% RSLogix 500 project alarm_count_live.RSS, saved by version 8.30.00.16 %
PROJECT "UNTITLED"    % processor: Bul.1763 MicroLogix 1100 Series B %

PROGRAM FILES
  LAD 2 "MAIN"  4 rungs
  LAD 3 "SUB_AND"  6 rungs
  LAD 4 "PARALLEL"  12 rungs
  LAD 5 "XIC_BRUTEF"  3 rungs
  LAD 6 "LOOKUPBYTE"  5 rungs
  LAD 7 "WRITE_BITS"  5 rungs
  LAD 255 "BITSPRBYTE"  5 rungs

DATA FILES
  O0 OUTPUT  4 elements
  I1 INPUT  6 elements
  S2 STATUS  66 elements
  B3 BINARY  3 elements
  T4 TIMER  11 elements
  C5 COUNTER  1 elements
  R6 CONTROL  1 elements
  N7 INTEGER  10 elements
  F8 FLOAT  4 elements
  L9 LONG_DATA  12 elements
  N10 BITSPRBYTE  256 elements
  L11 LONG_MASKS  12 elements
  L100 CONTRLTIME  256 elements
  L101 SUBANDTIME  256 elements
  L102 PARLLLTIME  256 elements
  L103 XIC_TIME  256 elements
  L104 LOOKUPTIME  256 elements

LADDER 2 "MAIN"
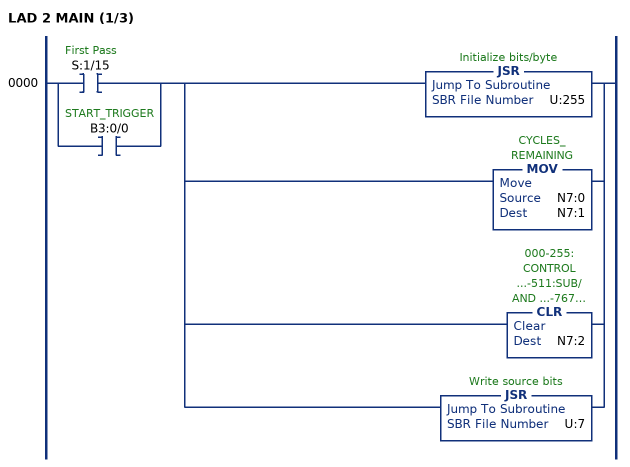
% Rung: 0 %
SOR BST XIC S:1/15 NXB XIC B3:0/0 BND BST JSR U:255 NXB MOV N7:0 N7:1 NXB CLR N7:2 NXB JSR U:7 BND EOR
%   S:1/15  "First Pass" %
%   B3:0/0  START_TRIGGER %
%   U:255  "Initialize bits/byte" %
%   N7:0  TEST_CYCLES %
%   N7:1  CYCLES_REMAINING %
%   N7:2  WHICH  "000-255:CONTROL ...-511:SUB/AND ...-767:PARALLEL ...-1023:XIC ...-1279:LOOKUP_BYTE" %
%   U:7  "Write source bits" %

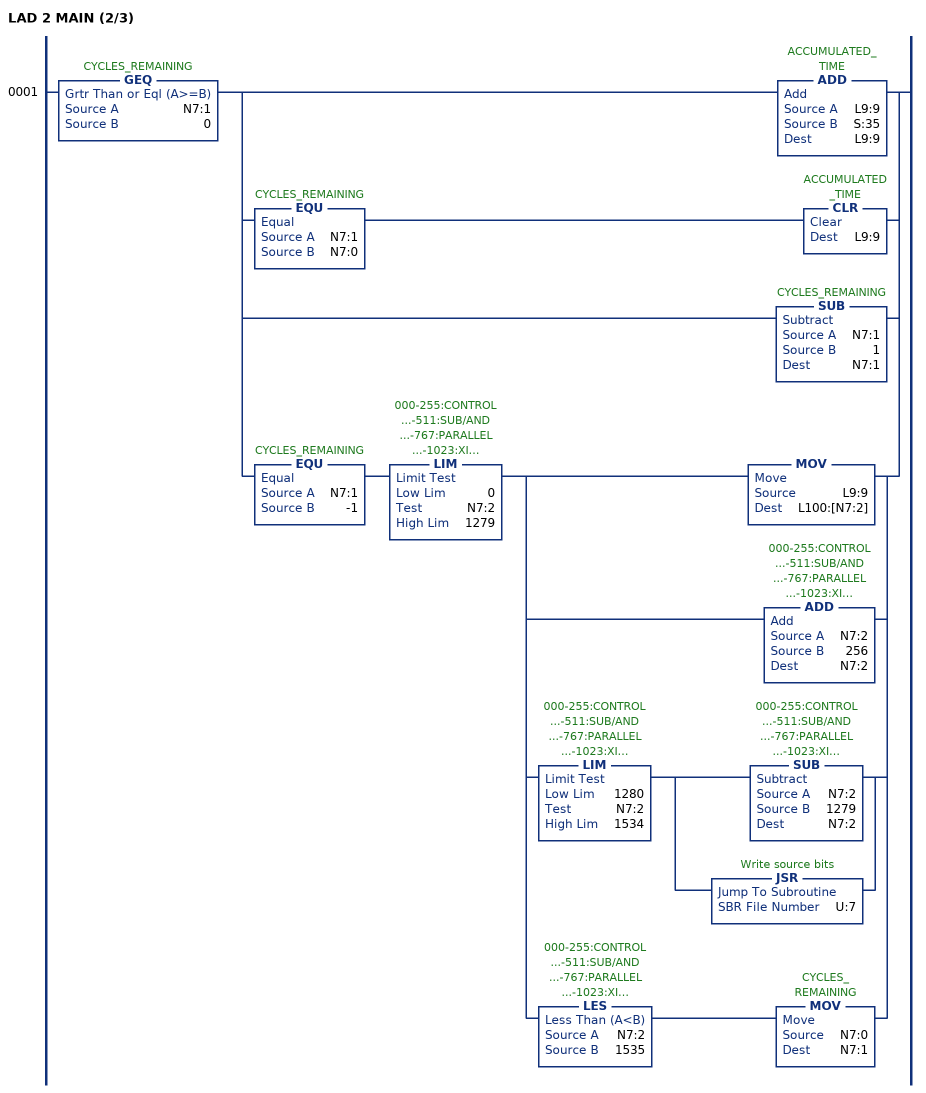
% Rung: 1 %
SOR GEQ N7:1 0 BST ADD L9:9 S:35 L9:9 NXB EQU N7:1 N7:0 CLR L9:9 NXB SUB N7:1 1 N7:1 NXB EQU N7:1 -1 LIM 0 N7:2 1279 BST MOV L9:9 L100:[N7:2] NXB ADD N7:2 256 N7:2 NXB LIM 1280 N7:2 1534 BST SUB N7:2 1279 N7:2 NXB JSR U:7 BND NXB LES N7:2 1535 MOV N7:0 N7:1 BND BND EOR
%   N7:1  CYCLES_REMAINING %
%   L9:9  ACCUMULATED_TIME %
%   S:35  "Last 1 ms Scan Time" %
%   N7:0  TEST_CYCLES %
%   N7:2  WHICH  "000-255:CONTROL ...-511:SUB/AND ...-767:PARALLEL ...-1023:XIC ...-1279:LOOKUP_BYTE" %
%   U:7  "Write source bits" %

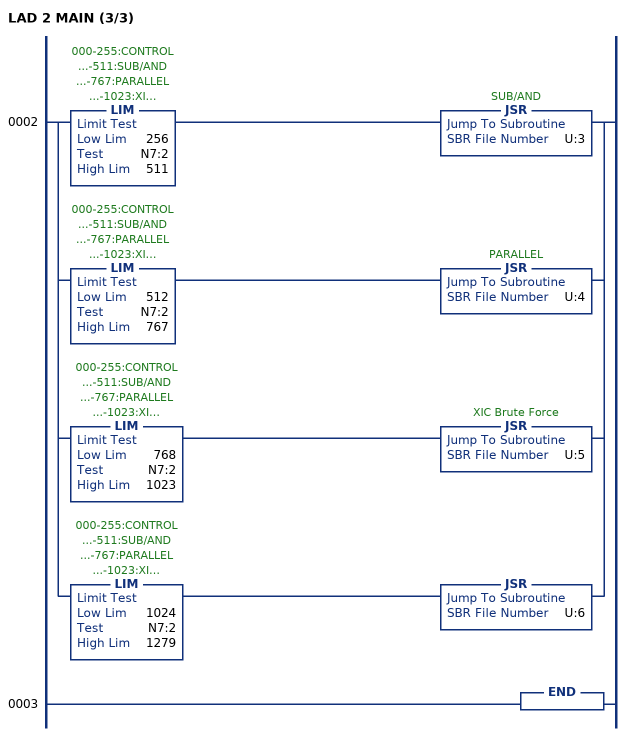
% Rung: 2 %
SOR BST LIM 256 N7:2 511 JSR U:3 NXB LIM 512 N7:2 767 JSR U:4 NXB LIM 768 N7:2 1023 JSR U:5 NXB LIM 1024 N7:2 1279 JSR U:6 BND EOR
%   N7:2  WHICH  "000-255:CONTROL ...-511:SUB/AND ...-767:PARALLEL ...-1023:XIC ...-1279:LOOKUP_BYTE" %
%   U:3  "SUB/AND" %
%   U:4  "PARALLEL" %
%   U:5  "XIC Brute Force" %
% Rung: 3 %
SOR END EOR

LADDER 3 "SUB_AND"
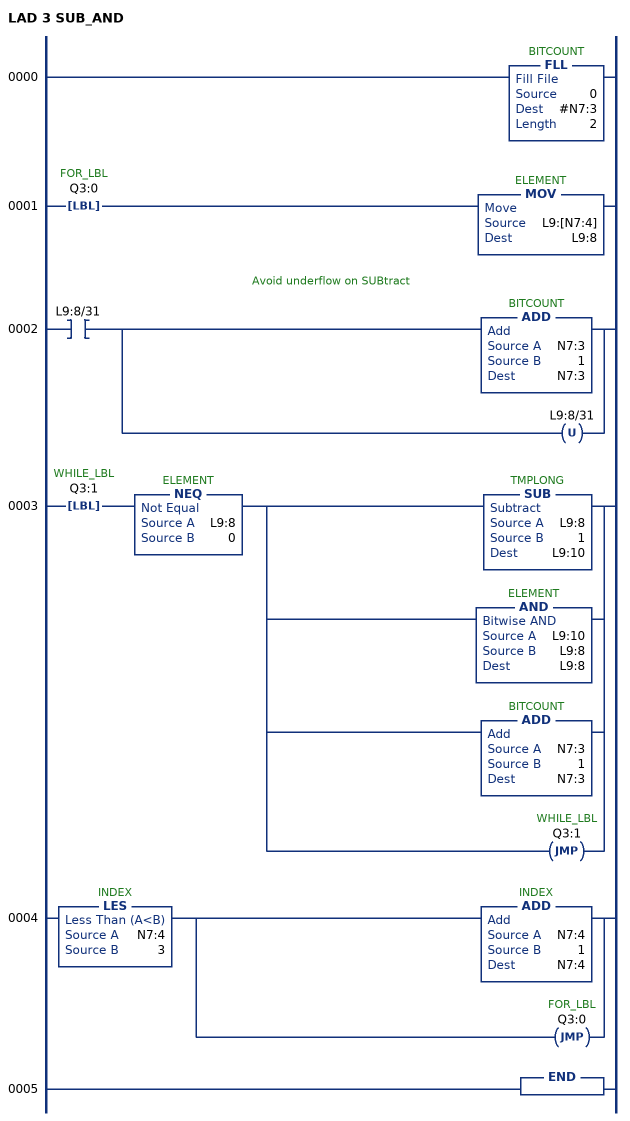
% Rung: 0 %
SOR FLL 0 #N7:3 2 EOR
%   N7:3  BITCOUNT %
% Rung: 1 %
SOR LBL Q3:0 MOV L9:[N7:4] L9:8 EOR
%   Q3:0  FOR_LBL %
%   N7:4  INDEX %
%   L9:8  ELEMENT %
% Rung: 2 %
% Avoid underflow on SUBtract %
SOR XIC L9:8/31 BST ADD N7:3 1 N7:3 NXB OTU L9:8/31 BND EOR
%   N7:3  BITCOUNT %
% Rung: 3 %
SOR LBL Q3:1 NEQ L9:8 0 BST SUB L9:8 1 L9:10 NXB AND L9:10 L9:8 L9:8 NXB ADD N7:3 1 N7:3 NXB JMP Q3:1 BND EOR
%   Q3:1  WHILE_LBL %
%   L9:8  ELEMENT %
%   L9:10  TMPLONG %
%   N7:3  BITCOUNT %
% Rung: 4 %
SOR LES N7:4 3 BST ADD N7:4 1 N7:4 NXB JMP Q3:0 BND EOR
%   N7:4  INDEX %
%   Q3:0  FOR_LBL %
% Rung: 5 %
SOR END EOR

LADDER 4 "PARALLEL"
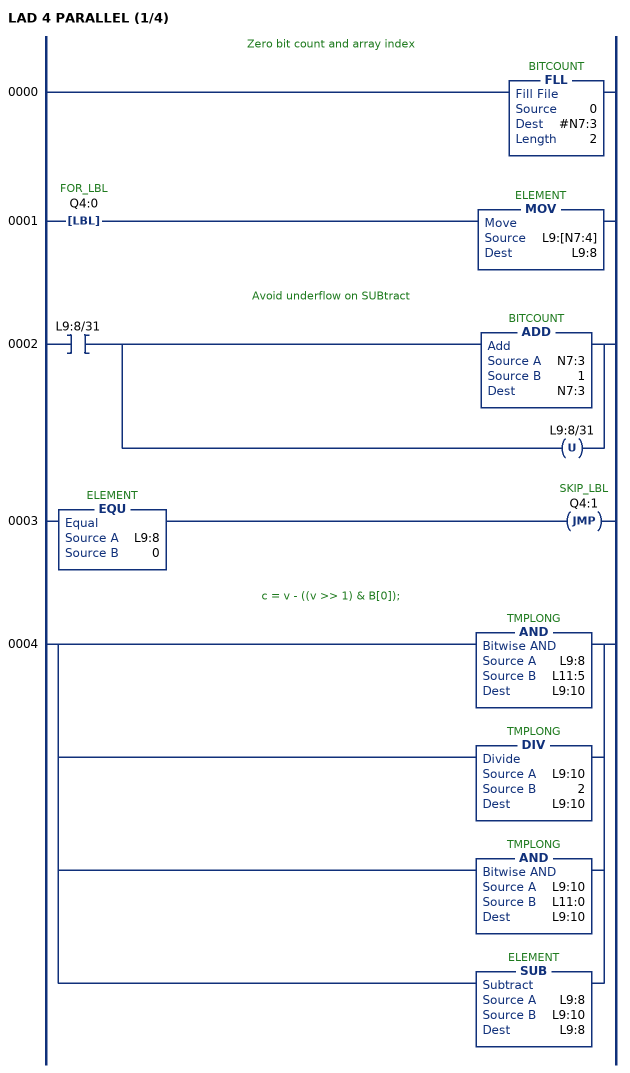
% Rung: 0 %
% Zero bit count and array index %
SOR FLL 0 #N7:3 2 EOR
%   N7:3  BITCOUNT %
% Rung: 1 %
SOR LBL Q4:0 MOV L9:[N7:4] L9:8 EOR
%   Q4:0  "FOR_LBL" %
%   N7:4  INDEX %
%   L9:8  ELEMENT %
% Rung: 2 %
% Avoid underflow on SUBtract %
SOR XIC L9:8/31 BST ADD N7:3 1 N7:3 NXB OTU L9:8/31 BND EOR
%   N7:3  BITCOUNT %
% Rung: 3 %
SOR EQU L9:8 0 JMP Q4:1 EOR
%   L9:8  ELEMENT %
%   Q4:1  "SKIP_LBL" %
% Rung: 4 %
% c = v - ((v >> 1) & B[0]); %
SOR BST AND L9:8 L11:5 L9:10 NXB DIV L9:10 2 L9:10 NXB AND L9:10 L11:0 L9:10 NXB SUB L9:8 L9:10 L9:8 BND EOR
%   L9:8  ELEMENT %
%   L11:5  0XFFFFFFFE_S0 %
%   L9:10  TMPLONG %
%   L11:0  0X55555555_B0 %

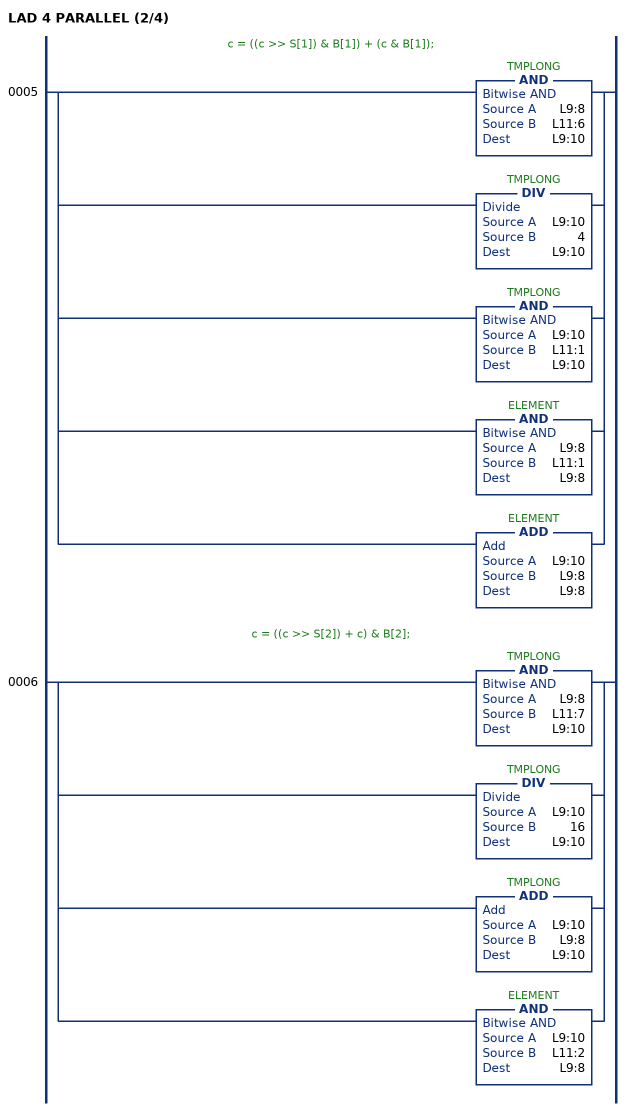
% Rung: 5 %
% c = ((c >> S[1]) & B[1]) + (c & B[1]); %
SOR BST AND L9:8 L11:6 L9:10 NXB DIV L9:10 4 L9:10 NXB AND L9:10 L11:1 L9:10 NXB AND L9:8 L11:1 L9:8 NXB ADD L9:10 L9:8 L9:8 BND EOR
%   L9:8  ELEMENT %
%   L11:6  0XFFFFFFFC_S1 %
%   L9:10  TMPLONG %
%   L11:1  0X33333333_B1 %
% Rung: 6 %
% c = ((c >> S[2]) + c) & B[2]; %
SOR BST AND L9:8 L11:7 L9:10 NXB DIV L9:10 16 L9:10 NXB ADD L9:10 L9:8 L9:10 NXB AND L9:10 L11:2 L9:8 BND EOR
%   L9:8  ELEMENT %
%   L11:7  0XFFFFFFF0_S2 %
%   L9:10  TMPLONG %
%   L11:2  0X0F0F0F0F_B2 %

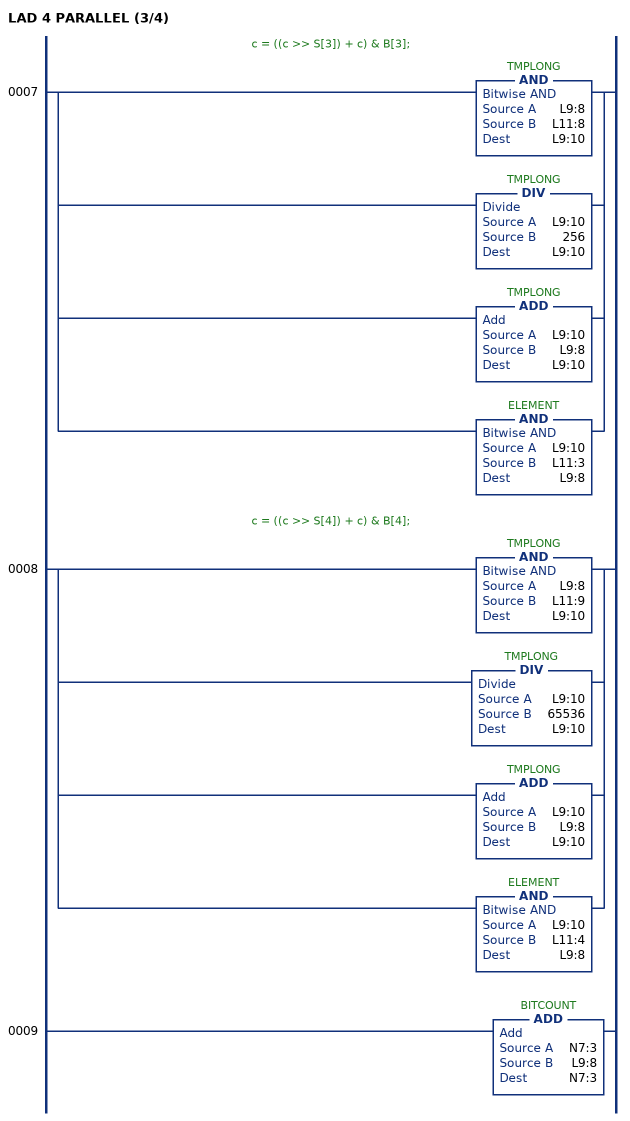
% Rung: 7 %
% c = ((c >> S[3]) + c) & B[3]; %
SOR BST AND L9:8 L11:8 L9:10 NXB DIV L9:10 256 L9:10 NXB ADD L9:10 L9:8 L9:10 NXB AND L9:10 L11:3 L9:8 BND EOR
%   L9:8  ELEMENT %
%   L11:8  0XFFFFFF00_S3 %
%   L9:10  TMPLONG %
%   L11:3  0X00FF00FF_B3 %
% Rung: 8 %
% c = ((c >> S[4]) + c) & B[4]; %
SOR BST AND L9:8 L11:9 L9:10 NXB DIV L9:10 65536 L9:10 NXB ADD L9:10 L9:8 L9:10 NXB AND L9:10 L11:4 L9:8 BND EOR
%   L9:8  ELEMENT %
%   L11:9  0XFFFF0000_S4 %
%   L9:10  TMPLONG %
%   L11:4  0X0000FFFF_B4 %
% Rung: 9 %
SOR ADD N7:3 L9:8 N7:3 EOR
%   N7:3  BITCOUNT %
%   L9:8  ELEMENT %

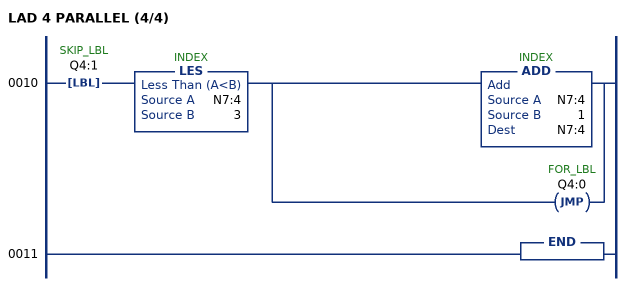
% Rung: 10 %
SOR LBL Q4:1 LES N7:4 3 BST ADD N7:4 1 N7:4 NXB JMP Q4:0 BND EOR
%   Q4:1  "SKIP_LBL" %
%   N7:4  INDEX %
%   Q4:0  "FOR_LBL" %
% Rung: 11 %
SOR END EOR

LADDER 5 "XIC_BRUTEF"
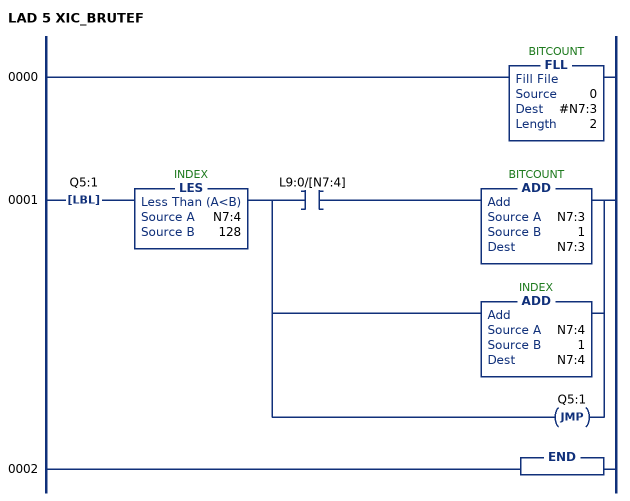
% Rung: 0 %
SOR FLL 0 #N7:3 2 EOR
%   N7:3  BITCOUNT %
% Rung: 1 %
SOR LBL Q5:1 LES N7:4 128 BST XIC L9:0/[N7:4] ADD N7:3 1 N7:3 NXB ADD N7:4 1 N7:4 NXB JMP Q5:1 BND EOR
%   N7:4  INDEX %
%   L9:0  128_SOURCE_BITS %
%   N7:3  BITCOUNT %
% Rung: 2 %
SOR END EOR

LADDER 6 "LOOKUPBYTE"
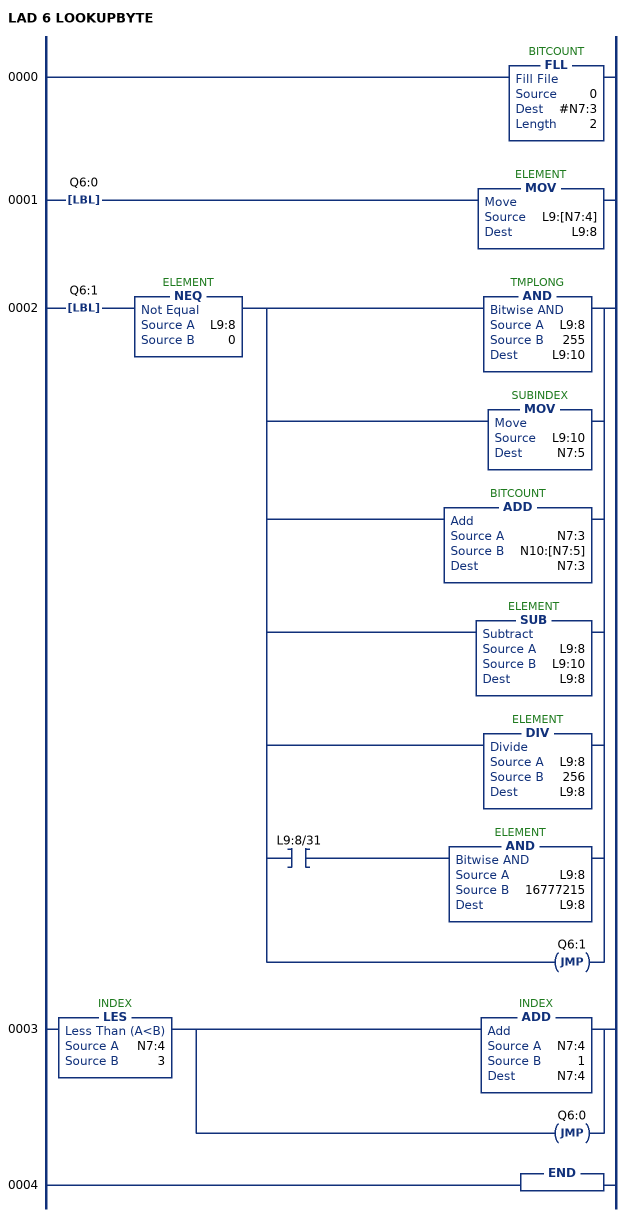
% Rung: 0 %
SOR FLL 0 #N7:3 2 EOR
%   N7:3  BITCOUNT %
% Rung: 1 %
SOR LBL Q6:0 MOV L9:[N7:4] L9:8 EOR
%   N7:4  INDEX %
%   L9:8  ELEMENT %
% Rung: 2 %
SOR LBL Q6:1 NEQ L9:8 0 BST AND L9:8 255 L9:10 NXB MOV L9:10 N7:5 NXB ADD N7:3 N10:[N7:5] N7:3 NXB SUB L9:8 L9:10 L9:8 NXB DIV L9:8 256 L9:8 NXB XIC L9:8/31 AND L9:8 16777215 L9:8 NXB JMP Q6:1 BND EOR
%   L9:8  ELEMENT %
%   L9:10  TMPLONG %
%   N7:5  SUBINDEX %
%   N7:3  BITCOUNT %
% Rung: 3 %
SOR LES N7:4 3 BST ADD N7:4 1 N7:4 NXB JMP Q6:0 BND EOR
%   N7:4  INDEX %
% Rung: 4 %
SOR END EOR

LADDER 7 "WRITE_BITS"
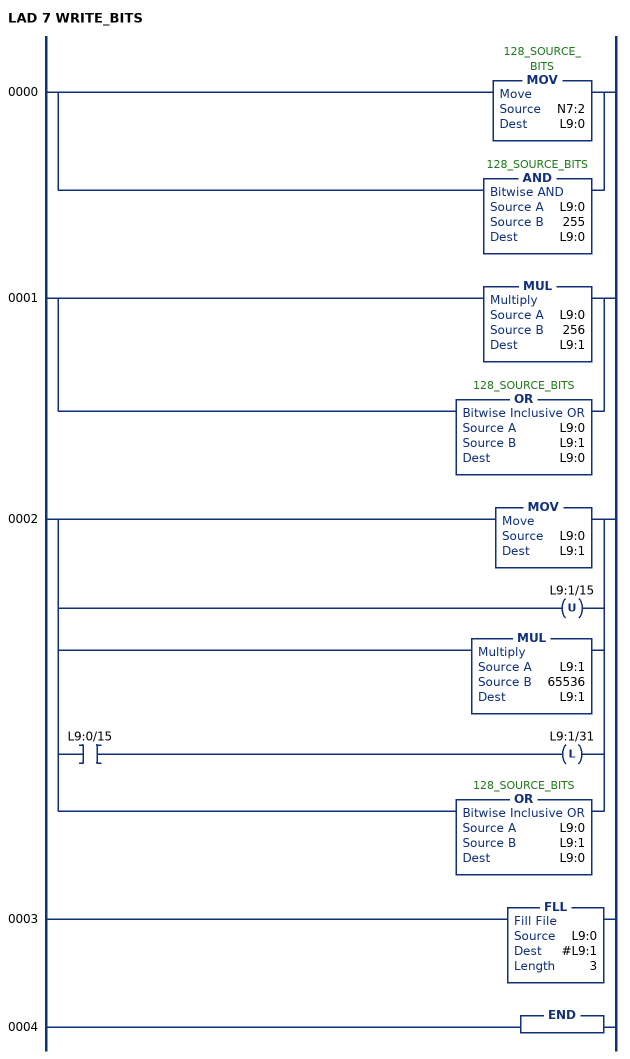
% Rung: 0 %
SOR BST MOV N7:2 L9:0 NXB AND L9:0 255 L9:0 BND EOR
%   N7:2  WHICH  "000-255:CONTROL ...-511:SUB/AND ...-767:PARALLEL ...-1023:XIC ...-1279:LOOKUP_BYTE" %
%   L9:0  128_SOURCE_BITS %
% Rung: 1 %
SOR BST MUL L9:0 256 L9:1 NXB OR L9:0 L9:1 L9:0 BND EOR
%   L9:0  128_SOURCE_BITS %
% Rung: 2 %
SOR BST MOV L9:0 L9:1 NXB OTU L9:1/15 NXB MUL L9:1 65536 L9:1 NXB XIC L9:0/15 OTL L9:1/31 NXB OR L9:0 L9:1 L9:0 BND EOR
%   L9:0  128_SOURCE_BITS %
% Rung: 3 %
SOR FLL L9:0 #L9:1 3 EOR
%   L9:0  128_SOURCE_BITS %
% Rung: 4 %
SOR END EOR

LADDER 255 "BITSPRBYTE"
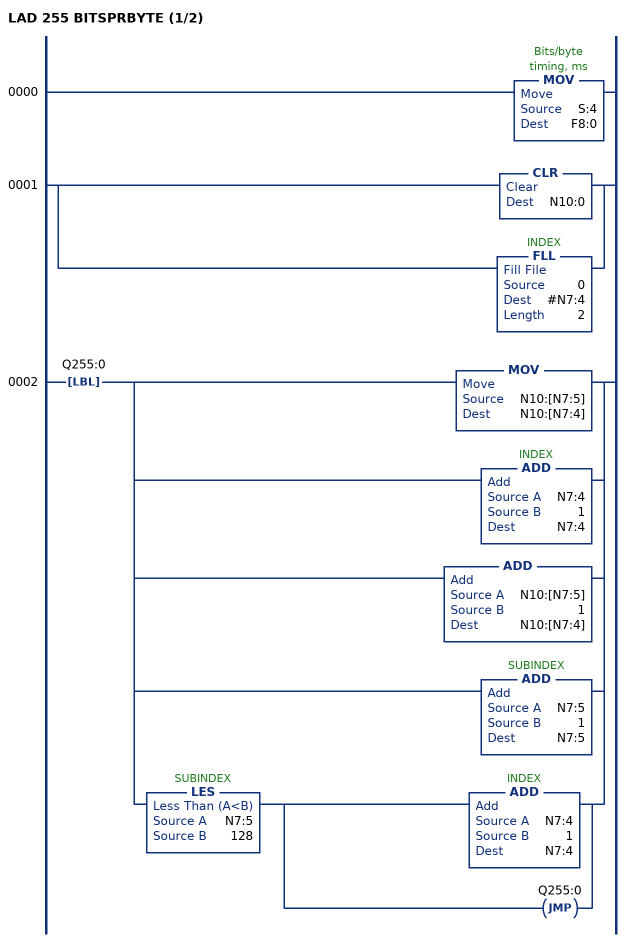
% Rung: 0 %
SOR MOV S:4 F8:0 EOR
%   S:4  "Time Base" %
%   F8:0  "Bits/byte timing, ms" %
% Rung: 1 %
SOR BST CLR N10:0 NXB FLL 0 #N7:4 2 BND EOR
%   N7:4  INDEX %
% Rung: 2 %
SOR LBL Q255:0 BST MOV N10:[N7:5] N10:[N7:4] NXB ADD N7:4 1 N7:4 NXB ADD N10:[N7:5] 1 N10:[N7:4] NXB ADD N7:5 1 N7:5 NXB LES N7:5 128 BST ADD N7:4 1 N7:4 NXB JMP Q255:0 BND BND EOR
%   N7:5  SUBINDEX %
%   N7:4  INDEX %

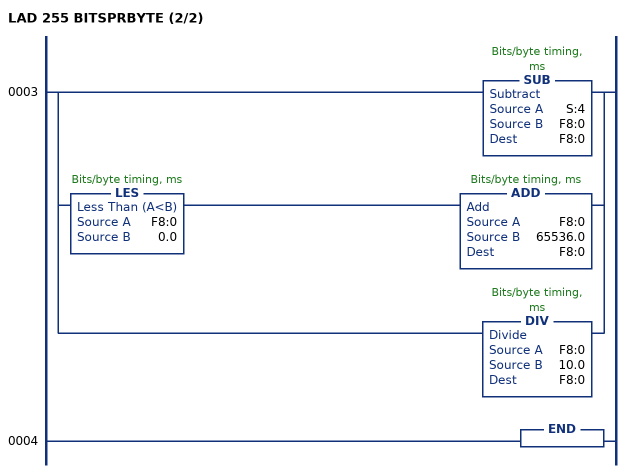
% Rung: 3 %
SOR BST SUB S:4 F8:0 F8:0 NXB LES F8:0 0.0 ADD F8:0 65536.0 F8:0 NXB DIV F8:0 10.0 F8:0 BND EOR
%   S:4  "Time Base" %
%   F8:0  "Bits/byte timing, ms" %
% Rung: 4 %
SOR END EOR

OTHER DOCUMENTED ADDRESSES
  L9:4  128_WORKING_BITS
  N7:6  8BITS

OTHER INSTRUCTION COMMENTS
  L9:4 NEQ  "First Working Long"

COMMENTS NOT ATTACHED TO A CURRENT RUNG
  N7:2/4: Restore preserved (cf. Rung 0005 above) bit values for /4 and /5

DATA TABLE (non-zero values as saved)
DATA T4
% .PRE .ACC %
% T4:1 % 5000 0
% T4:10 % 25 0
DATA C5
% .PRE .ACC %
% C5:0 % 1 0
DATA R6
% .LEN .POS %
% R6:0 % 128 0
DATA N7
% N7:0 % 1000 -1 1535 128 3 255 0 0 0 0
DATA F8
% F8:0 % 6.9 0 0 0
DATA L9
% L9:0 % -1 -1 -1 -1 0
% L9:5 % 0 0 0 0 19551
% L9:10 % 255 0
DATA N10
% N10:0 % 0 1 1 2 1 2 2 3 1 2
% N10:10 % 2 3 2 3 3 4 1 2 2 3
% N10:20 % 2 3 3 4 2 3 3 4 3 4
% N10:30 % 4 5 1 2 2 3 2 3 3 4
% N10:40 % 2 3 3 4 3 4 4 5 2 3
% N10:50 % 3 4 3 4 4 5 3 4 4 5
% N10:60 % 4 5 5 6 1 2 2 3 2 3
% N10:70 % 3 4 2 3 3 4 3 4 4 5
% N10:80 % 2 3 3 4 3 4 4 5 3 4
% N10:90 % 4 5 4 5 5 6 2 3 3 4
% N10:100 % 3 4 4 5 3 4 4 5 4 5
% N10:110 % 5 6 3 4 4 5 4 5 5 6
% N10:120 % 4 5 5 6 5 6 6 7 1 2
% N10:130 % 2 3 2 3 3 4 2 3 3 4
% N10:140 % 3 4 4 5 2 3 3 4 3 4
% N10:150 % 4 5 3 4 4 5 4 5 5 6
% N10:160 % 2 3 3 4 3 4 4 5 3 4
% N10:170 % 4 5 4 5 5 6 3 4 4 5
% N10:180 % 4 5 5 6 4 5 5 6 5 6
% N10:190 % 6 7 2 3 3 4 3 4 4 5
% N10:200 % 3 4 4 5 4 5 5 6 3 4
% N10:210 % 4 5 4 5 5 6 4 5 5 6
% N10:220 % 5 6 6 7 3 4 4 5 4 5
% N10:230 % 5 6 4 5 5 6 5 6 6 7
% N10:240 % 4 5 5 6 5 6 6 7 5 6
% N10:250 % 6 7 6 7 7 8
DATA L11
% L11:0 % 1431655765 858993459 252645135 16711935 65535
% L11:5 % -2 -4 -16 -256 -65536
DATA L100
% L100:0 % 8186 8718 8495 8523 8511
% L100:5 % 8517 8420 8361 8412 8374
% L100:10 % 8386 8391 8395 8384 8392
% L100:15 % 8381 8377 8392 8392 8367
% L100:20 % 8383 8401 8371 8377 8401
% L100:25 % 8406 8430 8390 8399 8389
% L100:30 % 8385 8392 8372 8390 8358
% L100:35 % 8389 8394 8382 8376 8380
% L100:40 % 8401 8369 8384 8399 8411
% L100:45 % 8390 8423 8403 8407 8408
% L100:50 % 8387 8393 8400 8407 8389
% L100:55 % 8376 8386 8381 8389 8373
% L100:60 % 8371 8396 7953 7971 7946
% L100:65 % 7961 7968 7965 7963 7968
% L100:70 % 7958 7961 7967 7937 7952
% L100:75 % 7953 7959 7937 7937 7945
% L100:80 % 7943 7948 7938 7938 7923
% L100:85 % 7940 7940 7936 7954 7940
% L100:90 % 7954 7942 7967 7961 7952
% L100:95 % 7966 7985 7971 7968 7969
% L100:100 % 7965 7965 7952 7943 7947
% L100:105 % 7943 8350 8380 8390 8380
% L100:110 % 8366 8366 8340 8370 8368
% L100:115 % 8369 8370 8405 8374 8384
% L100:120 % 8403 8399 8375 8360 8371
% L100:125 % 8344 8384 8362 8368 8379
% L100:130 % 8377 8366 8372 8390 8371
% L100:135 % 8379 8391 8385 8375 8366
% L100:140 % 8390 8353 8403 8366 8369
% L100:145 % 8386 8360 8375 8361 8368
% L100:150 % 8355 8361 8371 8371 8361
% L100:155 % 8380 8380 8393 8376 8394
% L100:160 % 8364 8379 8375 8380 8372
% L100:165 % 8378 8355 8362 8363 8353
% L100:170 % 8370 8358 8389 8367 8348
% L100:175 % 8368 8350 8343 8385 8381
% L100:180 % 8366 8387 8354 8372 8390
% L100:185 % 8369 8392 8381 8379 8377
% L100:190 % 8389 8387 8378 8364 8358
% L100:195 % 8364 8347 8369 8360 8363
% L100:200 % 8363 8362 8356 8369 8377
% L100:205 % 8370 8355 8366 8403 8377
% L100:210 % 8378 8382 8364 8362 8386
% L100:215 % 8349 8353 8372 8375 8362
% L100:220 % 8356 8361 8354 8383 8374
% L100:225 % 8376 8375 8404 8394 8375
% L100:230 % 8370 8370 8370 8357 8365
% L100:235 % 8347 8369 8359 8343 8355
% L100:240 % 8357 8389 8379 8361 8387
% L100:245 % 8374 8368 8400 8386 8362
% L100:250 % 8369 8364 8371 8365 8349
% L100:255 % 8366
DATA L101
% L101:0 % 10929 16432 15979 21431 16060
% L101:5 % 21436 21218 26593 15925 21190
% L101:10 % 21231 26498 21217 26539 26530
% L101:15 % 31844 15899 21240 21215 26562
% L101:20 % 21221 26522 26558 31847 21236
% L101:25 % 26507 26571 31798 26504 31847
% L101:30 % 31853 37138 15888 21240 21234
% L101:35 % 26538 21208 26560 26509 31863
% L101:40 % 21232 26513 26529 31806 26549
% L101:45 % 31824 31825 37158 21232 26517
% L101:50 % 26526 31843 26541 31827 31800
% L101:55 % 37114 26531 31866 31803 37109
% L101:60 % 31833 36114 35457 40504 15127
% L101:65 % 20197 20201 25298 20203 25285
% L101:70 % 25300 30352 20200 25286 25283
% L101:75 % 30356 25274 30355 30364 35439
% L101:80 % 20207 25285 25270 30340 25274
% L101:85 % 30354 30373 35434 25299 30361
% L101:90 % 30364 35435 30362 35427 35449
% L101:95 % 40512 20211 25292 25286 30370
% L101:100 % 25287 30367 30360 35443 25294
% L101:105 % 31830 31865 37129 31778 37093
% L101:110 % 37062 42341 26497 31835 31777
% L101:115 % 37092 31776 37102 37087 42381
% L101:120 % 31805 37068 37107 42347 37066
% L101:125 % 42380 42342 47664 14817 20107
% L101:130 % 20126 25419 20118 25434 25420
% L101:135 % 30742 20101 25417 25434 30735
% L101:140 % 25430 30721 30762 36031 20109
% L101:145 % 25442 25445 30756 25426 30730
% L101:150 % 30719 36029 25438 30749 30738
% L101:155 % 36060 30699 35985 36065 41311
% L101:160 % 20129 25433 25432 30774 25423
% L101:165 % 30722 30710 36024 25422 30762
% L101:170 % 30709 35973 30697 35961 35952
% L101:175 % 41261 25448 30748 30763 36035
% L101:180 % 30736 36030 36066 41264 30738
% L101:185 % 36042 36019 41258 36049 41297
% L101:190 % 41279 46563 20106 25454 25443
% L101:195 % 30746 25468 30706 30730 36020
% L101:200 % 25457 30740 30731 36015 30708
% L101:205 % 36028 36053 41316 25413 30696
% L101:210 % 30729 36042 30730 36050 36010
% L101:215 % 41286 30761 36023 36031 41290
% L101:220 % 36009 41249 41304 46598 25441
% L101:225 % 30752 30741 36053 30740 36025
% L101:230 % 36022 41303 30756 36009 36019
% L101:235 % 41267 36057 41308 41298 46584
% L101:240 % 30740 36017 36016 41298 35966
% L101:245 % 41320 41297 46599 36041 41309
% L101:250 % 41330 46522 41288 46573 46607
% L101:255 % 51882
DATA L102
% L102:0 % 10671 19300 18930 18902 18907
% L102:5 % 18946 18749 18743 18737 18696
% L102:10 % 18705 18724 18720 18711 18708
% L102:15 % 18700 18742 18709 18742 18738
% L102:20 % 18732 18726 18730 18736 18746
% L102:25 % 18725 18725 18736 18699 18726
% L102:30 % 18708 18746 18735 18726 18696
% L102:35 % 18700 18747 18722 18712 18718
% L102:40 % 18728 18710 18715 18727 18729
% L102:45 % 18741 18697 18724 18714 18742
% L102:50 % 18734 18692 18722 18740 18731
% L102:55 % 18733 18739 18733 18715 18750
% L102:60 % 18705 17843 17833 17838 17817
% L102:65 % 17837 17830 17813 17834 17826
% L102:70 % 17833 17827 17836 17827 17815
% L102:75 % 17819 17831 17834 17824 17828
% L102:80 % 17813 17834 17819 17794 17825
% L102:85 % 17829 17825 17831 17825 17832
% L102:90 % 17827 17834 17829 17833 17815
% L102:95 % 17831 17818 17835 17832 17824
% L102:100 % 17832 17824 17843 17817 17837
% L102:105 % 18929 18694 18704 18672 18705
% L102:110 % 18698 18699 18702 18691 18679
% L102:115 % 18706 18707 18690 18690 18680
% L102:120 % 18696 18698 18691 18709 18686
% L102:125 % 18687 18701 18697 18910 18976
% L102:130 % 18969 18936 18952 18955 18952
% L102:135 % 18951 18984 18967 18946 18953
% L102:140 % 18955 18966 18951 18969 18959
% L102:145 % 18976 18952 18952 18954 18976
% L102:150 % 18977 18964 18954 18970 18938
% L102:155 % 18941 18957 18964 18964 18983
% L102:160 % 18958 18977 18982 18959 18968
% L102:165 % 18960 18970 18960 18974 18943
% L102:170 % 18952 18974 18954 18953 18934
% L102:175 % 18972 18954 18982 18942 18976
% L102:180 % 18969 18978 18978 18958 18959
% L102:185 % 18952 18941 18979 18947 18966
% L102:190 % 18966 18964 18978 18964 18956
% L102:195 % 18952 18965 18982 18980 18949
% L102:200 % 18958 18957 18951 18949 18981
% L102:205 % 18956 18963 18976 18981 18972
% L102:210 % 18952 18971 18962 18980 18988
% L102:215 % 18955 18979 18967 18963 18942
% L102:220 % 18954 18972 18971 18944 18967
% L102:225 % 18970 18959 18929 18978 18952
% L102:230 % 18946 18970 18962 18976 18968
% L102:235 % 18932 18963 18955 18966 18953
% L102:240 % 18968 18987 18963 18946 18980
% L102:245 % 18972 18946 18945 18949 18943
% L102:250 % 18973 18959 18949 18963 18937
% L102:255 % 18960
DATA L103
% L103:0 % 38605 39684 39778 40864 39775
% L103:5 % 40684 40578 41681 39535 40574
% L103:10 % 40535 41630 40536 41594 41615
% L103:15 % 42723 39505 40560 40557 41617
% L103:20 % 40575 41559 41648 42687 40566
% L103:25 % 41606 41583 42569 41611 42635
% L103:30 % 42644 43713 39514 40570 40545
% L103:35 % 41625 40545 41586 41654 42659
% L103:40 % 40603 41651 41638 42684 41627
% L103:45 % 42645 42681 43674 40583 41609
% L103:50 % 41627 42450 41618 42648 42652
% L103:55 % 43720 41587 42629 42679 43834
% L103:60 % 42671 41794 41798 42813 37716
% L103:65 % 38739 38746 39741 38736 39743
% L103:70 % 39737 40754 38739 39736 39735
% L103:75 % 40756 39739 40759 40741 41765
% L103:80 % 38727 39720 39703 40705 39721
% L103:85 % 40779 40750 41766 39743 40760
% L103:90 % 40754 41772 40759 41768 41767
% L103:95 % 42807 38730 39741 39752 40743
% L103:100 % 39749 40762 40758 41765 39873
% L103:105 % 42668 42626 43665 42590 43650
% L103:110 % 43676 44730 41537 42592 42650
% L103:115 % 43692 42611 43663 43639 44653
% L103:120 % 42612 43670 43638 44706 43690
% L103:125 % 44737 44741 45808 39478 40497
% L103:130 % 40502 41566 40487 41542 41568
% L103:135 % 42572 40529 41511 41543 42627
% L103:140 % 41551 42623 42574 43620 40502
% L103:145 % 41548 41599 42573 41580 42626
% L103:150 % 42613 43641 41555 42628 42615
% L103:155 % 43671 42581 43677 43652 44718
% L103:160 % 40521 41576 41515 42586 41559
% L103:165 % 42587 42592 43659 41526 42598
% L103:170 % 42614 43656 42574 43627 43560
% L103:175 % 44730 41544 42630 42576 43679
% L103:180 % 42585 43642 43663 44753 42584
% L103:185 % 43709 43669 44675 43699 44721
% L103:190 % 44711 45761 40470 41530 41594
% L103:195 % 42615 41574 42630 42563 43683
% L103:200 % 41532 42606 42605 43683 42667
% L103:205 % 43646 43664 44731 41539 42586
% L103:210 % 42621 43675 42628 43672 43631
% L103:215 % 44653 42609 43654 43621 44694
% L103:220 % 43628 44685 44660 45812 41561
% L103:225 % 42629 42584 43674 42640 43643
% L103:230 % 43685 44693 42629 43691 43655
% L103:235 % 44683 43622 44732 44717 45793
% L103:240 % 42612 43666 43695 44686 43671
% L103:245 % 44689 44747 45757 43682 44692
% L103:250 % 44676 45735 44708 45746 45701
% L103:255 % 46835
DATA L104
% L104:0 % 10850 19529 19489 19580 19427
% L104:5 % 19301 19370 19375 19354 19338
% L104:10 % 19351 19343 19369 19357 19338
% L104:15 % 19329 19363 19344 19375 19381
% L104:20 % 19375 19378 19408 19376 19357
% L104:25 % 19383 19375 19376 19377 19368
% L104:30 % 19348 19364 19337 19363 19373
% L104:35 % 19353 19374 19361 19357 19342
% L104:40 % 19387 19366 19345 19370 19361
% L104:45 % 19376 19361 19379 19353 19362
% L104:50 % 19366 19360 19340 19352 19350
% L104:55 % 19358 19362 19368 19358 19500
% L104:60 % 19363 18449 18428 18433 18449
% L104:65 % 18426 18432 18440 18448 18435
% L104:70 % 18447 18437 18449 18444 18449
% L104:75 % 18442 18429 18431 18436 18429
% L104:80 % 18435 18415 18412 18412 18440
% L104:85 % 18425 18445 18426 18439 18432
% L104:90 % 18438 18428 18433 18436 18438
% L104:95 % 18424 18443 18427 18433 18441
% L104:100 % 18436 18440 18429 18445 18427
% L104:105 % 19405 19341 19338 19320 19345
% L104:110 % 19334 19349 19326 19336 19334
% L104:115 % 19370 19330 19326 19350 19323
% L104:120 % 19316 19351 19337 19332 19348
% L104:125 % 19322 19331 19327 19608 19595
% L104:130 % 19603 19604 19606 19598 19611
% L104:135 % 19570 19595 19585 19610 19600
% L104:140 % 19632 19598 19618 19600 19618
% L104:145 % 19619 19598 19596 19615 19595
% L104:150 % 19623 19614 19601 19620 19607
% L104:155 % 19642 19583 19614 19605 19609
% L104:160 % 19616 19609 19630 19589 19595
% L104:165 % 19633 19598 19631 19602 19588
% L104:170 % 19595 19574 19594 19577 19603
% L104:175 % 19617 19633 19574 19597 19601
% L104:180 % 19606 19601 19598 19592 19607
% L104:185 % 19621 19614 19596 19581 19592
% L104:190 % 19627 19595 19593 19601 19623
% L104:195 % 19612 19608 19608 19599 19621
% L104:200 % 19601 19622 19616 19609 19602
% L104:205 % 19637 19610 19605 19606 19586
% L104:210 % 19611 19593 19587 19577 19626
% L104:215 % 19621 19560 19609 19600 19605
% L104:220 % 19576 19623 19593 19609 19614
% L104:225 % 19608 19625 19608 19609 19592
% L104:230 % 19606 19577 19591 19619 19602
% L104:235 % 19592 19575 19613 19588 19575
% L104:240 % 19574 19587 19608 19612 19618
% L104:245 % 19582 19590 19588 19596 19607
% L104:250 % 19598 19586 19603 19607 19581
% L104:255 % 19551
